FUNCTION_BLOCK FBlock (* Basic function block *)
  (* Standard: 61499 *)
  (* Version 1.0, 11/20/2015 9:00 AM, Kawsihen, Kawsihen_s Macintosh *)
  (* Compiler header: package mypackage *)
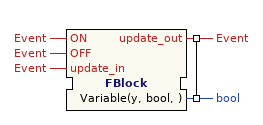
  EVENT_INPUT
    ON;
    OFF;
    update_in;
  END_EVENT
  EVENT_OUTPUT
    update_out WITH Variable(y, bool, );
  END_EVENT
  VAR_OUTPUT
    Variable(y, bool, ) : bool;
  END_VAR
  VAR
    k : REAL;
    d : REAL;
    x : REAL;
    C1x : REAL;
  END_VAR
  EC_STATES
    Start : init;
    t2 : t2Algo;
    t3 : t3Algo;
    t1 : t1Algo;
    t4 : t4Algo;
    t_state1 : t_state1Algo;
    t_state2 : t_state2Algo;
    t_state3 : t_state3Algo;
    t_state4 : t_state4Algo;
    t_state5 : t_state5Algo;
    t_state6 : t_state6Algo;
  END_STATES
  EC_TRANSITIONS
    Start TO t2 := True;
    t2 TO t_state1 := OFF;
    t_state1 TO t4 := True;
    t4 TO t_state2 := true &&  (x >= 20 && x <= 20);
    t_state2 TO t1 := True;
    t3 TO t_state3 := OFF;
    t_state3 TO t4 := True;
    t4 TO t_state4 := ON;
    t_state4 TO t2 := True;
    t1 TO t_state5 := ON;
    t_state5 TO t2 := True;
    t2 TO t_state6 := true &&  (x >= 100 && x <= 100);
    t_state6 TO t3 := True;
    t2 TO t2 := x >= 20 && x <= 100;
    t3 TO t3 := x >= 100 && x <= 100;
    t1 TO t1 := x >= 20 && x <= 20;
    t4 TO t4 := x >= 20 && x <= 100;
  END_TRANSITIONS
  ALGORITHM t2Algo IN C:
me->C1x = -130.00;
me->x = (float) me->C1x*exp(-0.075*me->d*me->k) + 150.0;
me->k++;
  END_ALGORITHM
  ALGORITHM t3Algo IN C:
me->C1x = 100.00;
me->x = (float) me->C1x;
me->k++;
  END_ALGORITHM
  ALGORITHM t1Algo IN C:
me->C1x = -50.000;
me->x = (float) me->C1x*exp(-0.075*me->d*me->k) + 150.0;
me->k++;
  END_ALGORITHM
  ALGORITHM t4Algo IN C:
me->C1x = 20.000;
me->x = (float) me->C1x;
me->k++;
  END_ALGORITHM
  ALGORITHM init IN C:
me->d = 0.01;
me->k = 0;
  END_ALGORITHM
  ALGORITHM t_state1Algo IN C:
me->k = 0;
  END_ALGORITHM
  ALGORITHM t_state2Algo IN C:
me->k = 0;
  END_ALGORITHM
  ALGORITHM t_state3Algo IN C:
me->k = 0;
  END_ALGORITHM
  ALGORITHM t_state4Algo IN C:
me->k = 0;
  END_ALGORITHM
  ALGORITHM t_state5Algo IN C:
me->k = 0;
  END_ALGORITHM
  ALGORITHM t_state6Algo IN C:
me->k = 0;
  END_ALGORITHM
END_FUNCTION_BLOCK
